TEXTLIST TextList_03
   = ''
END_TEXTLIST

(* stored: Version 1.1.0.1
   TextList TextList_03: Id {c2a0bda8-6316-0218-0e04-345d4ba82531} *)
